{attribute 'qualified_only'}
VAR_GLOBAL
	
	//fbPauseUI		:FB_SignalHandling :=(bSignalInput:= GVL_General.bPauseBtnUI);   cannot assigned the signal here.
	fbPauseUI		:FB_SignalHandling;
	
	fbHandleStartBtn		:FB_SignalHandling;
	inPauseBtnHandling		:FB_SignalHandling;
	inStopBtnHandling		:FB_SignalHandling;
END_VAR

(* stored: Version 1.1.0.1, ProductVersion 3.1.4022.16
   GVL GVL_SignalHanlding: Id {4ac69a16-daca-4fcb-9c6c-3f36991b4512} *)
